{attribute 'GeneratedUsingTerminal: EP7402-0057-0017'}
{attribute addProperty BoxType "EP7402-0057-0017"}
{attribute addProperty Id "InputAT %I*ARRAY[0..3] OF BOOL4Control_inputAT %I*ARRAY[0..3] OF BOOL4"}
{attribute addProperty CRC "56034484"}
{attribute addProperty Size "8"}
TYPE DI_Inputs_58955D1A :
STRUCT
	{attribute addProperty Name "Input"}
	Input AT %I* : ARRAY[0..3] OF BOOL;
	{attribute addProperty Name "Control_input"}
	Control_input AT %I* : ARRAY[0..3] OF BOOL;
END_STRUCT
END_TYPE

(* stored: Version 1.2.0.0, ProductVersion 3.1.4024.9
   DUT DI_Inputs_58955D1A: Id {3705f224-af4c-4293-8d0b-f27a48aed622} *)
